// TwinCAT 3 PLC project APRProject2i
// ProgramVersion: 3.1.4023.0
// libraries:
//   Tc2_Standard, * (Beckhoff Automation GmbH)
//   Tc2_System, * (Beckhoff Automation GmbH)
//   Tc3_Module, * (Beckhoff Automation GmbH)
// project tree:
//   DUTs/ sftDiModule.TcDUT, sftDoModule.TcDUT
//   / GlobalTextList.TcGTLO, PlcTask.TcTTO, Visualization Manager.TcVMO (not stored)
//   GVLs/ GVL.TcGVL, IO.TcGVL, VISU.TcGVL
//   POUs/ MAIN.TcPOU, sftDiCondAck.TcPOU, sftDiRunAck.TcPOU
//   VISUs/ StartVis.TcPOU, StartVisu.TcPOU, Visualization_1.TcVIS
// real-time tasks:
//   TASK PlcTask: cycle T#10ms, priority 20, ADS port 350
// I/O:
//   DEVICE Device 1 (Beckhoff CCAT)
//   DEVICE Device 2 (EtherCAT), AmsNetId 5.52.95.234.3.1
//     Term 1 (EK1200) [EK1200-5000 EtherCAT Power supply (2A E-Bus)]
//       Term 2 (EL2008) [EL2008 8Ch. Dig. Output 24V, 0.5A]
//       Term 3 (EL2008) [EL2008 8Ch. Dig. Output 24V, 0.5A]
//       Term 4 (EL4021) [EL4021 1Ch. Ana. Output 4-20mA, 12bit]
//       Term 5 (EL4021) [EL4021 1Ch. Ana. Output 4-20mA, 12bit]
//       Term 6 (EL3021) [EL3021 1Ch. Ana. Input 4-20mA DIFF]
//       Term 7 (EL2008) [EL2008 8Ch. Dig. Output 24V, 0.5A]
//       Box 8 (BK1250)
// variable links:
//   APRProject2i/APRProject2i Instance <-> Device 2 (EtherCAT)/Term 1 (EK1200)/Box 8 (BK1250)
//     PlcTask Inputs/IO.f2_REF <-> Term 6 (KL3102)/Channel 1/IO.f2_REF
//     PlcTask Inputs/IO.f3_REF <-> Term 6 (KL3102)/Channel 2/IO.f3_REF
//     PlcTask Inputs/IO.f4_REF <-> Term 7 (KL3102)/Channel 1/IO.f4_REF
//     PlcTask Outputs/IO.k2_REF <-> Term 3 (KL4132)/Channel 2/IO.k2_REF
//     PlcTask Outputs/IO.k3_REF <-> Term 2 (KL4132)/Channel 2/IO.k3_REF
//     PlcTask Outputs/IO.k4_REF <-> Term 4 (KL4132)/Channel 2/IO.k4_REF
//   APRProject2i/APRProject2i Instance <-> Device 2 (EtherCAT)/Term 1 (EK1200)/Term 2 (EL2008)
//     PlcTask Outputs/IO.r{1..6}_REF <-> Channel {1..6}/Output  (6 links)
//     PlcTask Outputs/IO.v1_REF <-> Channel 7/Output
//     PlcTask Outputs/IO.v2_REF <-> Channel 8/Output
//   APRProject2i/APRProject2i Instance <-> Device 2 (EtherCAT)/Term 1 (EK1200)/Term 4 (EL4021)
//     PlcTask Outputs/IO.k1_REF <-> AO Outputs/IO.k1_REF
//   APRProject2i/APRProject2i Instance <-> Device 2 (EtherCAT)/Term 1 (EK1200)/Term 6 (EL3021)
//     PlcTask Inputs/IO.f1_REF <-> AI Standard/IO.f1_REF
//   APRProject2i/APRProject2i Instance <-> Device 2 (EtherCAT)/Term 1 (EK1200)/Term 7 (EL2008)
//     PlcTask Outputs/IO.fx{1..8}_REF <-> Channel {1..8}/Output  (8 links)

CONFIGURATION APRProject2i
    RESOURCE PLC ON TwinCAT3
        TASK PlcTask(INTERVAL := T#10ms, PRIORITY := 20);
        PROGRAM MAIN WITH PlcTask : MAIN;
    END_RESOURCE
END_CONFIGURATION

// ---- DUTs/sftDiModule.TcDUT
TYPE sftDiModule :
STRUCT
	sftDiRunVE1: 							io.p1_REF;
	sftDiRunVE2:  			 				io.p2_REF;
	sftDiRunVE3:  							io.p3_REF;
	sftDiRunVE4:  			 				io.p4_REF;
END_STRUCT
END_TYPE

// ---- DUTs/sftDoModule.TcDUT
TYPE sftDoModule :
STRUCT
	sftDoRunVE1: 			 				io.r1_REF;
	sftDoRunVE2:  			 				io.r2_REF;
	sftDoRunVE3:  							io.r3_REF;
	sftDoRunVE4:  			 				io.r4_REF;
	
	
END_STRUCT
END_TYPE

// ---- GVLs/GVL.TcGVL
{attribute 'qualified_only'}
VAR_GLOBAL



	
	
END_VAR

// ---- GVLs/IO.TcGVL
{attribute 'qualified_only'}
VAR_GLOBAL
	(* *) (* *) (* *) (* *) (* *) (* *) (* *) (* *) (* *) (* *) (* *) (* *) (* *)
	QualAck AT %I*:BOOL:=TRUE;
	(* *) (* *) (* *) (* *) (* *) (* *) (* *) (* *) (* *) (* *) (* *) (* *) (* *)
	p1_REF AT %I* : BOOL := FALSE; (*non-formal format: used with all dirxd*)
	p2_REF AT %I* : BOOL := FALSE; 
	p3_REF AT %I* : BOOL := FALSE;
	p4_REF AT %I* : BOOL := FALSE; 
	p5_REF AT %I* : BOOL := FALSE; 
	(* *) (* *) (* *) (* *) (* *) (* *) (* *) (* *) (* *) (* *) (* *) (* *) (* *)
	erikoismuuttujaSum AT %I* : BOOL := FALSE; 
	erikoismuuttujaDev AT %I* : BOOL := FALSE; 
	(* *) (* *) (* *) (* *) (* *) (* *) (* *) (* *) (* *) (* *) (* *) (* *) (* *)
	r1_REF AT %Q* : BOOL := FALSE; (*non-formal format: used with all dotxd*)
	r2_REF AT %Q* : BOOL := FALSE; 
	r3_REF AT %Q* : BOOL := FALSE;
	r4_REF AT %Q* : BOOL := FALSE; 
	r5_REF AT %Q* : BOOL := FALSE; (*non-formal format: used with all dotxd*)
	r6_REF AT %Q* : BOOL := FALSE; 
	(* *) (* *) (* *) (* *) (* *) (* *) (* *) (* *) (* *) (* *) (* *) (* *) (* *)
	fx1_REF AT %Q* : BOOL := FALSE; (* FMC 12 VDC BOOL 1|0 *) 
	fx2_REF AT %Q* : BOOL := FALSE; (* FMC 12 VDC BOOL 1|0 *) 
	fx3_REF AT %Q* : BOOL := FALSE; (* FMC 12 VDC BOOL 1|0 *) 
	fx4_REF AT %Q* : BOOL := FALSE; (* FMC 12 VDC BOOL 1|0 *) 
	fx5_REF AT %Q* : BOOL := FALSE; (* FMC 12 VDC BOOL 1|0 *) 
	fx6_REF AT %Q* : BOOL := FALSE; (* FMC 12 VDC BOOL 1|0 *) 
	fx7_REF AT %Q* : BOOL := FALSE; (* FMC 12 VDC BOOL 1|0 *) 
	fx8_REF AT %Q* : BOOL := FALSE; (* FMC 12 VDC BOOL 1|0 *) 	
	 (* *) (* *) (* *) (* *) (* *) (* *) (* *) (* *) (* *) (* *) (* *) (* *) (* *)
	v1_REF AT %Q* : BOOL := FALSE;
	v2_REF AT %Q* : BOOL := FALSE; 
	(* *) (* *) (* *) (* *) (* *) (* *) (* *) (* *) (* *) (* *) (* *) (* *) (* *)
	f1_REF AT %I*: INT; (* measured value (analog output for FMC, analog input for terminal, page 15) *) 
	f2_REF AT %I*: INT; (* measured value (analog output for FMC, analog input for terminal, page 15) *) 
	f3_REF AT %I*: INT; (* measured value (analog output for FMC, analog input for terminal, page 15) *) 
	f4_REF AT %I*: INT; (* measured value (analog output for FMC, analog input for terminal, page 15) *) 
	f5_REF AT %I*: INT; (* measured value (analog output for FMC, analog input for terminal, page 15) *) 
	(* *) (* *) (* *) (* *) (* *) (* *) (* *) (* *) (* *) (* *) (* *) (* *) (* *)
	(* *) (* *) (* *) (* *) (* USER INPUT *) (* *) (* *) (* *) (* *) (* *) (* *) 	
	UI1_REF : INT; // default = 31 IF scale = 15633 (* setpoint analog input for FMC, analog output for terminal, page 15) *)
	UI2_REF : INT; // default = 31 IF scale = 15633 (* setpoint analog input for FMC, analog output for terminal, page 15) *)
	UI3_REF : INT; // default = 31 IF scale = 15633 (* setpoint analog input for FMC, analog output for terminal, page 15) *)
	UI4_REF : INT; // default = 31 IF scale = 15633 (* setpoint analog input for FMC, analog output for terminal, page 15) *)
	UI5_REF : INT; // default = 31 IF scale = 15633 (* setpoint analog input for FMC, analog output for terminal, page 15) *)
	(* *) (* *) (* *) (* *) (* CONVERSION *) (* *) (* *) (* *) (* *) (* *) (* *) 	
//	c1_REF : INT :=31; // default = 31 IF scale = 15633 (* setpoint analog input for FMC, analog output for terminal, page 15) *)
//	c2_REF : INT :=31; // default = 31 IF scale = 15633 (* setpoint analog input for FMC, analog output for terminal, page 15) *)
//	c3_REF : INT :=31; // default = 31 IF scale = 15633 (* setpoint analog input for FMC, analog output for terminal, page 15) *)
//	c4_REF : INT :=31; // default = 31 IF scale = 15633 (* setpoint analog input for FMC, analog output for terminal, page 15) *)
//	c5_REF : INT :=31; // default = 31 IF scale = 15633 (* setpoint analog input for FMC, analog output for terminal, page 15) *)
	(* *) (* *) (* *) (* *) (* *) (* *) (* *) (* *) (* *) (* *) (* *) (* *) (* *)
	k1_REF AT %Q*: INT; (* setpoint analog input for FMC, analog output for terminal, page 15) *)
	k2_REF AT %Q*: INT; (* setpoint analog input for FMC, analog output for terminal, page 15) *)
	k3_REF AT %Q*: INT; (* setpoint analog input for FMC, analog output for terminal, page 15) *)
	k4_REF AT %Q*: INT; (* setpoint analog input for FMC, analog output for terminal, page 15) *)
	k5_REF AT %Q*: INT; (* setpoint analog input for FMC, analog output for terminal, page 15) *)
	(* *) (* *) (* *) (* *) (* *) (* *) (* *) (* *) (* *) (* *) (* *) (* *) (* *)

	
	
	
	
	 // INT 15633 ja flow 30 ml/min 
	
	(* assign to term 3 KL3102 DATA IN *)

	
	

	


END_VAR

// ---- GVLs/VISU.TcGVL
{attribute 'qualified_only'}
VAR_GLOBAL
	
	bRunning: BOOL;	
	sState :STRING; (*tilatietoa, 80 merkkiä, muutoin string(255) jolloin merkkien pituus 255*)
// yksi merkki on aina yksi byte


END_VAR

// ---- POUs/MAIN.TcPOU
PROGRAM MAIN
VAR
	(* *) (* *) (* *) (* *) (* *) (* *) (* *) (* *) (* *) (* *) (* *) (* *) (* *)
	meter1: INT;
	meter2: INT;	
	meter3: INT;	
	meter4: INT;	
	meter5: INT;	
	(* *) (* *) (* *) (* *) (* *) (* *) (* *) (* *) (* *) (* *) (* *) (* *) (* *)
	idx: BOOL;
	idxDev: BOOL;
	(* *) (* *) (* *) (* *) (* *) (* *) (* *) (* *) (* *) (* *) (* *) (* *) (* *)
END_VAR
VAR
END_VAR

(*
start item = [] consist of fx1,fx2,fx3,fx4,fx5 and are assigned to output terminals 
meter = [] sample consists of metrics conversions from LREAL TO INT and loses some information
io.pX_REF = [] sample commandsio.p1_REF,io.p2_REF,io.p3_REF,io.p4_REF,io.p5_REF vars interconnected to ->
IF -loop where when assigned True enables IO variable write to io.k1_REF,io.k2_REF,io.k3_REF,io.k4_REF,io.k5_REF
in which assigned vars are INTs and enable to control flow directly from the terminal output to item input. 
*)
(* *) (* *) (* *) (* *) (* *) (* *) (* *) (* *) (* *) (* *) (* *) (* *) (* *)
(* *) (* *) (* *) (* *) (* *) (* *) (* *) (* *) (* *) (* *) (* *) (* *) (* *)
(* *) (* *) (* *) (* *) (* *) (* *) (* *) (* *) (* *) (* *) (* *) (* *) (* *)
(* *) (* *) (* *) (* *) (* *) (* *) (* *) (* *) (* *) (* *) (* *) (* *) (* *)
(* *) (* *) (* *) (* *) (* *) (* *) (* *) (* *) (* *) (* *) (* *) (* *) (* *)
(* *) (* *) (* *) (* *) (* *) (* *) (* *) (* *) (* *) (* *) (* *) (* *) (* *)
(* *) (* *) (* *) (* *) (* *) (* *) (* *) (* *) (* *) (* *) (* *) (* *) (* *)
(* *) (* *) (* *) (* *) (* *) (* *) (* *) (* *) (* *) (* *) (* *) (* *) (* *)
(* *) (* *) (* *) (* *) (* *) (* *) (* *) (* *) (* *) (* *) (* *) (* *) (* *)
(* *) (* *) (* *) (* *) (* CURRENT CONTROL *) (* *) (* *) (* *) (* *) (* *)
IF IO.p1_REF = TRUE THEN
	IO.k1_REF:=10000;
	ELSE
		IO.k1_REF:=0;	
END_IF
(* *) (* *) (* *) (* *) (* VOLTAGE CONTROL *) (* *) (* *) (* *) (* *) (* *)
IF IO.p2_REF = TRUE THEN
	IO.k2_REF:=10000;
	ELSE
		IO.k2_REF:=0;	
END_IF
(* *) (* *) (* *) (* *) (* VOLTAGE CONTROL *) (* *) (* *) (* *) (* *) (* *)
IF IO.p3_REF = TRUE THEN
	IO.k3_REF:=10000;
	ELSE
		IO.k3_REF:=0;	
END_IF
(* *) (* *) (* *) (* *) (* VOLTAGE CONTROL *) (* *) (* *) (* *) (* *) (* *)
IF IO.p4_REF = TRUE THEN
	IO.k4_REF:=10000;
	ELSE
		IO.k4_REF:=0;	
END_IF
(* *) (* *) (* *) (* *) (* VOLTAGE CONTROL *) (* *) (* *) (* *) (* *) (* *)
IF IO.p5_REF = TRUE THEN
	IO.k5_REF:=10000;
	ELSE
		IO.k5_REF:=0;	
END_IF
(* *) (* *) (* *) (* *) (* *) (* *) (* *) (* *) (* *) (* *) (* *) (* *) (* *)
(* *) (* *) (* *) (* *) (* *) (* *) (* *) (* *) (* *) (* *) (* *) (* *) (* *)
(* *) (* *) (* *) (* *) (* *) (* *) (* *) (* *) (* *) (* *) (* *) (* *) (* *)
(* *) (* *) (* *) (* *) (* *) (* *) (* *) (* *) (* *) (* *) (* *) (* *) (* *)
(* *) (* *) (* *) (* *) (* *) (* *) (* *) (* *) (* *) (* *) (* *) (* *) (* *)
(* *) (* *) (* *) (* *) (* *) (* *) (* *) (* *) (* *) (* *) (* *) (* *) (* *)
(* *) (* *) (* *) (* *) (* *) (* *) (* *) (* *) (* *) (* *) (* *) (* *) (* *)
(* *) (* *) (* *) (* *) (* *) (* *) (* *) (* *) (* *) (* *) (* *) (* *) (* *)
IF IO.p1_REF = TRUE THEN
	IO.k1_REF:=10000;
	ELSE
		IO.k1_REF:=0;	
END_IF
(* *) (* *) (* *) (* *) (* *) (* *) (* *) (* *) (* *) (* *) (* *) (* *) (* *)
(* *) (* *) (* *) (* *) (* *) (* *) (* *) (* *) (* *) (* *) (* *) (* *) (* *)
(* *) (* *) (* *) (* *) (* *) (* *) (* *) (* *) (* *) (* *) (* *) (* *) (* *)
(* *) (* *) (* *) (* *) (* *) (* *) (* *) (* *) (* *) (* *) (* *) (* *) (* *)
(* *) (* *) (* *) (* *) (* CLOSES ALL VALVES *) (* *) (* *) (* *) (* *) (* *)
IF IO.erikoismuuttujaSum=TRUE OR io.r1_REF =TRUE AND io.r2_REF =TRUE AND io.r3_REF =TRUE AND io.r4_REF =TRUE AND io.r5_REF =TRUE AND io.r6_REF =TRUE AND io.v1_REF =TRUE AND io.v2_REF =TRUE AND idx =TRUE THEN
		idx:=TRUE;
	io.r1_REF:=TRUE;
	io.r2_REF:=TRUE;	
			io.r3_REF:=TRUE;
	io.r4_REF:=TRUE;
			io.r5_REF:=TRUE;
	io.r6_REF:=TRUE;
			io.v1_REF:=TRUE;
	io.v2_REF:=TRUE;
	END_IF
(* *) (* *) (* *) (* *) (* *) (* *) (* *) (* *) (* *) (* *) (* *) (* *) (* *)
(* *) (* *) (* *) (* *) (* *) (* *) (* *) (* *) (* *) (* *) (* *) (* *) (* *)
(* *) (* *) (* *) (* *) (* *) (* *) (* *) (* *) (* *) (* *) (* *) (* *) (* *)
(* *) (* *) (* *) (* *) (* *) (* *) (* *) (* *) (* *) (* *) (* *) (* *) (* *)
(* *) (* *) (* *) (* *) (* KEEPS VALVES CLOSED *) (* *) (* *) (* *) (* *) (* *)
IF IO.erikoismuuttujaSum=FALSE AND idx=TRUE THEN
	idx:=FALSE;
			io.r1_REF:=FALSE;
	io.r2_REF:=FALSE;
			io.r3_REF:=FALSE;
	io.r4_REF:=FALSE;
			io.r5_REF:=FALSE;
	io.r6_REF:=FALSE;
			io.v1_REF:=FALSE;
	io.v2_REF:=FALSE;
END_IF
(* *) (* *) (* *) (* *) (* *) (* *) (* *) (* *) (* *) (* *) (* *) (* *) (* *)
///////////////////////////////////////////////////////////////////////////
(* *) (* *) (* *) (* *) (* *) (* *) (* *) (* *) (* *) (* *) (* *) (* *) (* *)
///////////////////////////////////////////////////////////////////////////
(* *) (* *) (* *) (* *) (* *) (* *) (* *) (* *) (* *) (* *) (* *) (* *) (* *)
(*CONVERTS LREAL ITEM OUTPUTS INTO TERMINAL INPUTS OF INT OF REAL WORLD SCALE*)
meter1:=io.UI1_REF; (*25 ml/min*) (*/819.5*100*); //ADD CONVERSION // AGD ? CURRENT
meter2:=io.f2_REF/65; (*25 ml/min*) (*/819.5*100*); //ADD CONVERSION // VOLTAGE
meter3:=io.f3_REF/65; (*25 ml/min*) (*/819.5*100*); //ADD CONVERSION // VOLTAGE
meter4:=io.f4_REF;//65 (*25 ml/min*) (*/819.5*100*); //ADD CONVERSION // VOLTAGE
meter5:=io.f5_REF;//520 (*25 ml/min*) (*/819.5*100*); //ADD CONVERSION // VOLTAGE
// k1_REF AS OVERRIDING ODD INPUT VALUES
// 
// meter1:=io.k1_REF/31 (* N ml/min *) (*/819.5*100*); //ADD CONVERSION // AGD ? CURRENT
// meter2:=io.k2_REF/31 (* N ml/min *) (*/819.5*100*); //ADD CONVERSION // VOLTAGE
// meter3:=io.k3_REF/31 (* N ml/min *) (*/819.5*100*); //ADD CONVERSION // VOLTAGE
// meter4:=io.k4_REF/31 (* N ml/min *) (*/819.5*100*); //ADD CONVERSION // VOLTAGE
// meter5:=io.k5_REF/31 (* N ml/min *) (*/819.5*100*); //ADD CONVERSION // VOLTAGE
//  
(* *) (* *) (* *) (* *) (* *) (* *) (* *) (* *) (* *) (* *) (* *) (* *) (* *)
(* *) (* *) (* *) (* *) (* *) (* *) (* *) (* *) (* *) (* *) (* *) (* *) (* *)
(* *) (* *) (* *) (* *) (* *) (* *) (* *) (* *) (* *) (* *) (* *) (* *) (* *)
(* *) (* *) (* *) (* *) (* *) (* *) (* *) (* *) (* *) (* *) (* *) (* *) (* *)
(* *) (* *) (* *) (* *) (* *) (* *) (* *) (* *) (* *) (* *) (* *) (* *) (* *)
(* *) (* *) (* *) (* *) (* *) (* *) (* *) (* *) (* *) (* *) (* *) (* *) (* *)
(* *) (* *) (* *) (* *) (* *) (* *) (* *) (* *) (* *) (* *) (* *) (* *) (* *)
(*CONVERTS LREAL ITEM OUTPUTS INTO TERMINAL INPUTS OF INT OF REAL WORLD SCALE*)
io.k1_REF:=65*io.UI1_REF;  (*25 ml/min*) (*/819.5*100*); //ADD CONVERSION // VOLTAGE //OK
io.k2_REF:=65*io.UI2_REF; //30 (*25 ml/min*) (*/819.5*100*); //ADD CONVERSION // VOLTAGE //
io.k3_REF:=65*io.UI3_REF;  (*25 ml/min*) (*/819.5*100*); //ADD CONVERSION // VOLTAGE //
io.k4_REF:=65*io.UI4_REF;  (*25 ml/min*) (*/819.5*100*); //ADD CONVERSION // VOLTAGE //
io.k5_REF:=30*io.UI5_REF;  (*25 ml/min*) (*/819.5*100*); //ADD CONVERSION // VOLTAGE //
(* *) (* *) (* *) (* *) (* *) (* *) (* *) (* *) (* *) (* *) (* *) (* *) (* *)
(* *) (* *) (* *) (* *) (* *) (* *) (* *) (* *) (* *) (* *) (* *) (* *) (* *)
(* *) (* *) (* *) (* *) (* *) (* *) (* *) (* *) (* *) (* *) (* *) (* *) (* *)
(* *) (* *) (* *) (* *) (* *) (* *) (* *) (* *) (* *) (* *) (* *) (* *) (* *)
(* *) (* *) (* *) (* *) (* *) (* *) (* *) (* *) (* *) (* *) (* *) (* *) (* *)



IF visu.bRunning=TRUE THEN
	VISU.sState := 'running';
ELSE
	VISU.sState := 'stopped';
END_IF




IF io.fx1_REF=FALSE THEN
	meter1:=0; (*25 ml/min*) (*/819.5*100*); //ADD CONVERSION // AGD ? CURRENT
	meter2:=0; (*25 ml/min*) (*/819.5*100*); //ADD CONVERSION // VOLTAGE
	meter3:=0; (*25 ml/min*) (*/819.5*100*); //ADD CONVERSION // VOLTAGE
	meter4:=0;//65 (*25 ml/min*) (*/819.5*100*); //ADD CONVERSION // VOLTAGE
	meter5:=0;//520 (*25 ml/min*) (*/819.5*100*); //ADD CONVERSION // VOLTAGE
	io.UI1_REF:=0;
	io.UI2_REF:=0;
	io.UI3_REF:=0;
	io.UI4_REF:=0;
	io.UI5_REF:=0;
ELSIF io.fx1_REF=FALSE THEN
	meter1:=io.UI1_REF; (*25 ml/min*) (*/819.5*100*); //ADD CONVERSION // AGD ? CURRENT
	meter2:=io.f2_REF; (*25 ml/min*) (*/819.5*100*); //ADD CONVERSION // VOLTAGE
	meter3:=io.f3_REF; (*25 ml/min*) (*/819.5*100*); //ADD CONVERSION // VOLTAGE
	meter4:=io.f4_REF;//65 (*25 ml/min*) (*/819.5*100*); //ADD CONVERSION // VOLTAGE
	meter5:=io.f5_REF;//520 (*25 ml/min*) (*/819.5*100*); //ADD CONVERSION // VOLTAGE
	io.k1_REF:=65*io.UI1_REF;  (*25 ml/min*) (*/819.5*100*); //ADD CONVERSION // VOLTAGE //OK
	io.k2_REF:=65*io.UI2_REF;  (*25 ml/min*) (*/819.5*100*); //ADD CONVERSION // VOLTAGE //
	io.k3_REF:=65*io.UI3_REF;  (*25 ml/min*) (*/819.5*100*); //ADD CONVERSION // VOLTAGE //
	io.k4_REF:=65*io.UI4_REF;  (*25 ml/min*) (*/819.5*100*); //ADD CONVERSION // VOLTAGE //
	io.k5_REF:=30*io.UI5_REF;  (*25 ml/min*) (*/819.5*100*); //ADD CONVERSION // VOLTAGE //
END_IF

END_PROGRAM

// ---- POUs/sftDiCondAck.TcPOU
FUNCTION_BLOCK sftDiCondAck
VAR
END_VAR
VAR_INPUT
	mcbutB1:=sftDiModule.sftDiRunVE1;
	mcbutB2:=sftDiModule.sftDiRunVE2;
	mcbutB3:=sftDiModule.sftDiRunVE3;
	mcbutB4:=sftDiModule.sftDiRunVE4;
END_VAR
VAR
END_VAR
VAR_OUTPUT
	sentREF1: BOOL;
	sentREF2: BOOL;
	sentREF3: BOOL;
	sentREF4: BOOL;
END_VAR
VAR
END_VAR

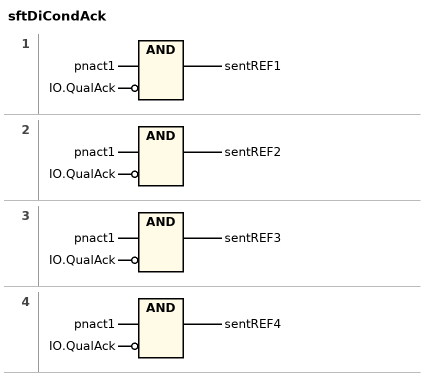
// NETWORK 1
sentREF1 := pnact1 AND NOT IO.QualAck;

// NETWORK 2
sentREF2 := pnact1 AND NOT IO.QualAck;

// NETWORK 3
sentREF3 := pnact1 AND NOT IO.QualAck;

// NETWORK 4
sentREF4 := pnact1 AND NOT IO.QualAck;

END_FUNCTION_BLOCK

// ---- POUs/sftDiRunAck.TcPOU
FUNCTION_BLOCK sftDiRunAck
VAR_INPUT
	sftDiRunIntrinsic1:sftDiCondAck;
	sftDiRunIntrinsic2:sftDiCondAck;	
	sftDiRunIntrinsic3:sftDiCondAck;
	sftDiRunIntrinsic4:sftDiCondAck;
END_VAR

VAR_OUTPUT	
	pnact1:=sftDoModule.sftDoRunVE1;
	pnact2:=sftDoModule.sftDoRunVE2;
	pnact3:=sftDoModule.sftDoRunVE3;
	pnact4:=sftDoModule.sftDoRunVE4;
END_VAR
VAR
END_VAR

sftDiRunIntrinsic1(sftDiModule.sftDiRunVE1:= IO.QualAck, sentREF1=> sftDoModule.sftDoRunVE1);
sftDiRunIntrinsic2(sftDiModule.sftDiRunVE2:= IO.QualAck, sentREF1=> sftDoModule.sftDoRunVE2);
sftDiRunIntrinsic3(sftDiModule.sftDiRunVE3:= IO.QualAck, sentREF1=> sftDoModule.sftDoRunVE3);
sftDiRunIntrinsic4(sftDiModule.sftDiRunVE4:= IO.QualAck, sentREF1=> sftDoModule.sftDoRunVE4);

END_FUNCTION_BLOCK

// ---- VISUs/StartVis.TcPOU
PROGRAM StartVis
VAR
	NT_StartProcess_0: NT_StartProcess;
	
END_VAR

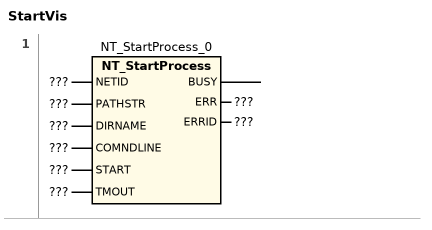
// NETWORK 1
NT_StartProcess_0(); // NT_StartProcess

END_PROGRAM

// ---- VISUs/StartVisu.TcPOU
PROGRAM StartVisu

VAR_INPUT
    NETID     : T_AmsNetId;
    PATHSTR   : T_MaxString;
    DIRNAME   : T_MaxString;
    COMNDLINE : T_MaxString;
    START     : BOOL;
    TMOUT     : TIME := DEFAULT_ADS_TIMEOUT;
END_VAR



VAR
END_VAR

END_PROGRAM

// ---- GlobalTextList.TcGTLO
TEXTLIST GlobalTextList
  440 = ''
  770 = "'ON/OFF ALL VALVES'"
  993 = "'ON/OFF FCs'"
  239 = "'OPEN/CLOSE VE1'"
  1 = "'OPEN/CLOSE VE4'"
  906 = "'OPEN/CLOSE VP1'"
  423 = "'OPEN/CLOSE VP2'"
  138 = "'OPEN/CLOSE VP3'"
  125 = "'OPEN/CLOSE VP4'"
  21 = "'OPEN/CLOSE VP5'"
  182 = "'OPEN/CLOSE VP6'"
  745 = '1st el2001 in order of terminals from 1 to 8.'
  373 = '1ST EL2001 TERMINALS FROM 1 TO 8 IN ORDER'
  424 = 'el2001 in order of terminals from 1 to 8.'
  318 = 'FLOW-COMMAND TOOL 2020'
  565 = 'FMC1 norm.clos.'
  452 = 'FMC2 norm.open'
  252 = 'FMC3 norm.clos.'
  590 = 'FMC4 norm.clos.'
  93 = 'ML/MIN'
  986 = 'norm clos'
  659 = 'norm open'
  897 = 'norm open toim.'
  941 = 'norm open?'
  716 = 'TERMINALS FROM 1 TO 8 IN ORDER (1ST EL2001) '
  599 = 'TERMINALS FROM 1 TO 8 IN ORDER 1ST EL2001 '
  121 = 'testaamat'
END_TEXTLIST

// ---- VISUs/Visualization_1.TcVIS
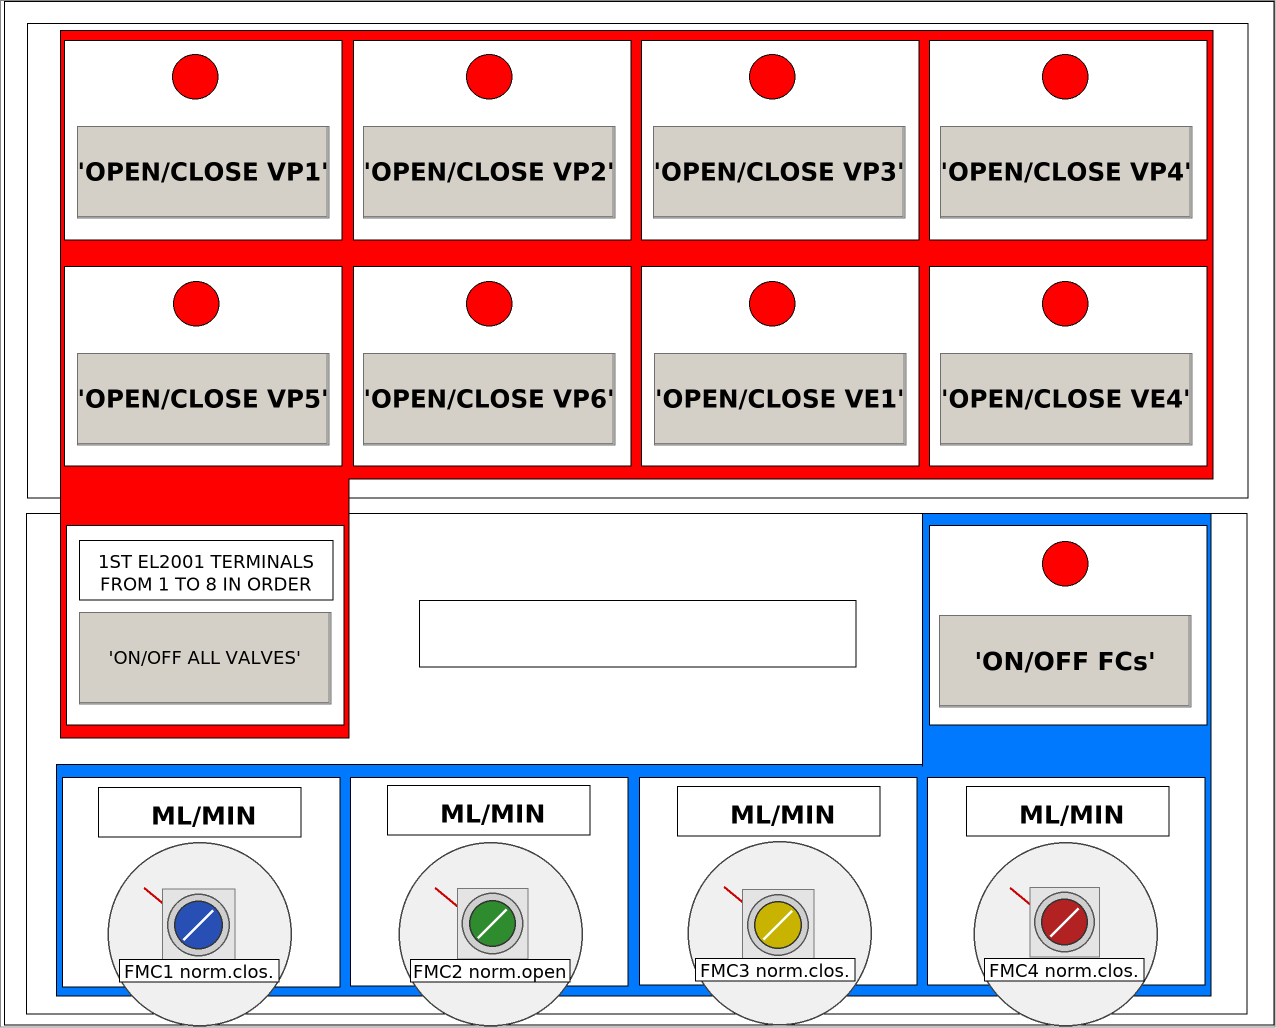
VISUALIZATION Visualization_1  // 1276x1028
    Rectangle (4,1 1270x1024)
    Rectangle (26,513 1221x501)
    Rectangle (56,764 1155x232)
    Rectangle (27,23 1221x475)
    RoundedRectangle (350,777 278x209)
    RoundedRectangle (62,777 278x210)
    RoundedRectangle (927,777 278x208)
    RoundedRectangle (639,777 278x208)
    Meter180 (104,842 191x184), value: MAIN.meter1, style: Meter-Meter180-Blue, scale format: %.1f, scale 0..500
    Potentiometer360 (162,886 73x78), variable: io.UI1_REF, style: Potentiometer-Potentiometer360-Blue, scale 0..500
        p2431819421: Outside
    Meter180 (395,842 191x184), value: MAIN.meter2, style: Meter-Meter180-Green, scale format: %.1f, scale 0..500
    Potentiometer360 (454,888 77x71), variable: io.UI2_REF, style: Potentiometer-Potentiometer360-Green, scale 0..500
        p2431819421: Outside
    Meter180 (684,841 191x184), value: MAIN.meter3, style: Meter-Meter180-Yellow, scale format: %.1f, scale 0..500
    Potentiometer360 (742,885 72x80), variable: io.UI3_REF, style: Potentiometer-Potentiometer360-Yellow, scale 0..500
        p2431819421: Outside
    Meter180 (970,842 191x184), value: MAIN.meter4, style: Meter-Meter180-Red, scale format: %.1f, scale 0..500
    Potentiometer360 (1029,887 71x70), variable: io.UI4_REF, style: Potentiometer-Potentiometer360-Red, scale 0..500
        p2431819421: Outside
    RoundedRectangle (98,787 203x50), text variable: meter1
    Textfield (123,795 162x41), "ML/MIN", text variable: MAIN.meter1
    RoundedRectangle (387,785 203x50)
    Textfield (412,793 162x41), "ML/MIN", text variable: MAIN.meter2
    RoundedRectangle (677,786 203x50)
    Textfield (702,794 162x41), "ML/MIN", text variable: MAIN.meter3
    RoundedRectangle (966,786 203x50)
    Textfield (991,794 162x41), "ML/MIN", text variable: MAIN.meter4
    RoundedRectangle (419,600 437x67)
    Label (392,588 495x92), "FLOW-COMMAND TOOL 2020"
    Rectangle (922,513 289x253)
    RoundedRectangle (929,525 278x200)
    Ellipse (1042,541 46x45), colour toggle: IO.fx1_REF
    Button (939,615 252x92), "'ON/OFF FCs'"
        OnMouseClick: toggle IO.fx1_REF
        OnMouseClick: toggle IO.fx2_REF
        OnMouseClick: toggle IO.fx3_REF
        OnMouseClick: toggle IO.fx4_REF
        OnMouseClick: toggle IO.fx5_REF
        OnMouseClick: toggle IO.fx6_REF
        OnMouseClick: toggle IO.fx7_REF
        OnMouseClick: toggle IO.fx8_REF
    Rectangle (60,477 289x261)
    Ellipse (181,536 46x45), colour toggle: IO.erikoismuuttujaSum
    RoundedRectangle (66,525 278x200)
    Button (79,612 252x92), "'ON/OFF ALL VALVES'"
        OnMouseClick: toggle IO.erikoismuuttujaSum
    Rectangle (60,30 1153x449)
    RoundedRectangle (353,266 278x200)
    RoundedRectangle (64,266 278x200)
    RoundedRectangle (353,40 278x200)
    RoundedRectangle (64,40 278x200)
    Ellipse (172,54 46x45), colour toggle: IO.r1_REF
    Button (77,126 252x92), "'OPEN/CLOSE VP1'"
        OnMouseClick: toggle IO.r1_REF
    Ellipse (466,54 46x45), colour toggle: IO.r2_REF
    Button (363,126 252x92), "'OPEN/CLOSE VP2'"
        OnMouseClick: toggle IO.r2_REF
    Ellipse (173,281 46x45), colour toggle: IO.r5_REF
    Button (77,353 252x92), "'OPEN/CLOSE VP5'"
        OnMouseClick: toggle IO.r5_REF
    Ellipse (466,281 46x45), colour toggle: IO.r6_REF
    Button (363,353 252x92), "'OPEN/CLOSE VP6'"
        OnMouseClick: toggle IO.r6_REF
    RoundedRectangle (929,266 278x200)
    RoundedRectangle (641,266 278x200)
    RoundedRectangle (929,40 278x200)
    RoundedRectangle (641,40 278x200)
    Ellipse (749,54 46x45), colour toggle: IO.r3_REF
    Button (653,126 252x92), "'OPEN/CLOSE VP3'"
        OnMouseClick: toggle IO.r3_REF
    Ellipse (1042,54 46x45), colour toggle: IO.r4_REF
    Button (940,126 252x92), "'OPEN/CLOSE VP4'"
        OnMouseClick: toggle IO.r4_REF
    Ellipse (749,281 46x45), colour toggle: IO.v1_REF
    Button (654,353 252x92), "'OPEN/CLOSE VE1'"
        OnMouseClick: toggle IO.v1_REF
    Ellipse (1042,281 46x45), colour toggle: IO.v2_REF
    Button (940,353 252x92), "'OPEN/CLOSE VE4'"
        OnMouseClick: toggle IO.v2_REF
    Rectangle (61,468 287x41)
    Rectangle (923,735 287x41)
    RoundedRectangle (119,959 160x23), text variable: meter1
    Textfield (120,963 158x18), "FMC1 norm.clos.", text variable: MAIN.meter3
    RoundedRectangle (410,959 160x23), text variable: meter1
    Textfield (411,963 158x18), "FMC2 norm.open", text variable: MAIN.meter3
    RoundedRectangle (695,958 160x23), text variable: meter1
    Textfield (696,962 158x18), "FMC3 norm.clos.", text variable: MAIN.meter3
    RoundedRectangle (984,958 160x23), text variable: meter1
    Textfield (985,962 158x18), "FMC4 norm.clos.", text variable: MAIN.meter3
    RoundedRectangle (79,540 254x60), text variable: meter1
    Textfield (80,549 252x48), "1ST EL2001 TERMINALS FROM 1 TO 8 IN ORDER", text variable: MAIN.meter3
END_VISUALIZATION
